FUNCTION printChangeAxisEnable : BOOL
VAR_INPUT
	cmd: ChangeAxisEnable;
END_VAR
VAR
END_VAR

MSG.changeAxisEnable.ipArguments.Clear().AddInt(cmd.axisIndex).AddBool(cmd.enabled);
MSG.changeAxisEnable.Send(0);

END_FUNCTION

(* stored: Version 1.1.0.1, ProductVersion 3.1.4022.12
   POU printChangeAxisEnable: Id {66b8293d-95cd-4d7e-946a-cbeedec012cf}, SpecialFunc None *)
